// TIA Portal V17 export
// export: Created 2023-12-22T15:28:36.9333419Z, ExportSetting WithDefaults, DisplayName Totally Integrated Automation Portal, DisplayVersion V17, DisplayName TIA Portal Openness, DisplayVersion V17, DisplayName TIA Portal Version Control Interface, DisplayVersion V17, DisplayName STEP 7 Professional, DisplayVersion V17, DisplayName STEP 7 Safety, DisplayVersion V17, DisplayName WinCC Advanced, DisplayVersion V17
DATA_BLOCK "Valves_DB"   // DB250
VERSION : 0.1
// stored: AutoNumber false, DBAccessibleFromOPCUA true, InstanceOfName Valves, InstanceOfType FB
"Valves"
   // VAR RETAIN
   //    Time_DTL { S7_SetPoint := 'True'} : DTL;
   // END_VAR
BEGIN
END_DATA_BLOCK
